{attribute 'qualified_only'}
{attribute 'strict'}
{attribute 'to_string'}
TYPE eCoolingSystemState :
(
	OFF 						:= 	0,
	Circulating					:=	1,
	ActiveCooling				:= 	2,
	ActiveHeating				:= 	3,
	EMSTOP						:=	5
)uint := OFF;
END_TYPE

(* stored: Version 1.1.0.1, ProductVersion 3.1.4026.18
   DUT eCoolingSystemState: Id {3d9938d8-59c8-4bba-9c8e-5ac8a873a19e} *)
